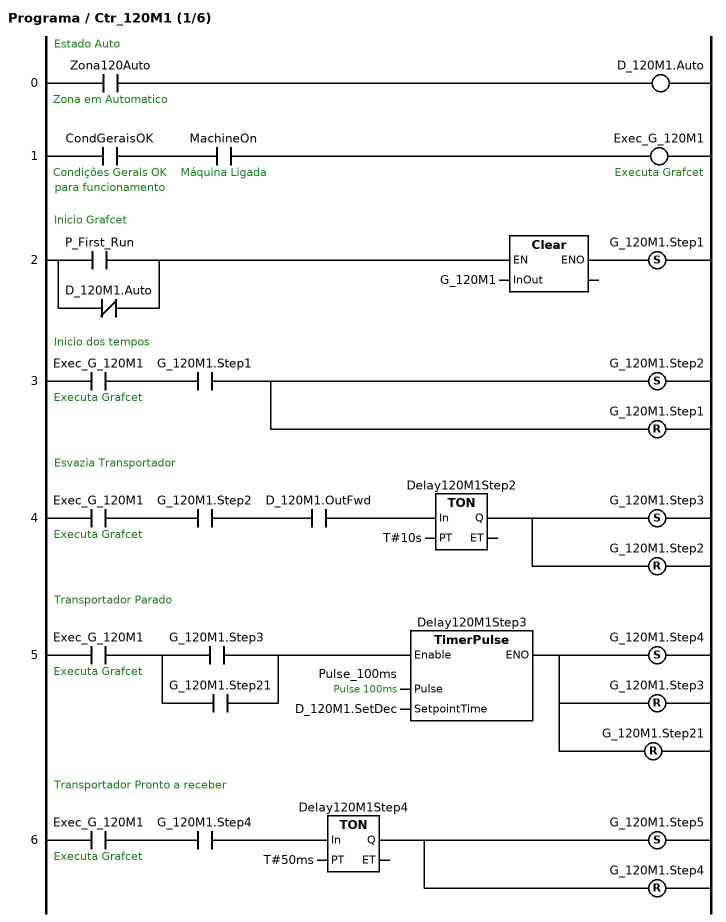
(* [picture p24: Programa / Ctr_120M1, rungs 0-6] *)
(* Rung 0: Estado Auto *)
D_120M1.Auto := Zona120Auto;
(* Rung 1 *)
Exec_G_120M1 := CondGeraisOK AND MachineOn;
(* Rung 2: Inicio Grafcet *)
IF P_First_Run OR NOT D_120M1.Auto THEN
    Clear(InOut := G_120M1);
    G_120M1.Step1 := TRUE;
END_IF;
(* Rung 3: Inicio dos tempos *)
_p41 := Exec_G_120M1 AND G_120M1.Step1;
IF _p41 THEN
    G_120M1.Step2 := TRUE;
    G_120M1.Step1 := FALSE;
END_IF;
(* Rung 4: Esvazia Transportador *)
Delay120M1Step2(In := Exec_G_120M1 AND G_120M1.Step2 AND D_120M1.OutFwd, PT := T#10s);
IF Delay120M1Step2.Q THEN
    G_120M1.Step3 := TRUE;
    G_120M1.Step2 := FALSE;
END_IF;
(* Rung 5: Transportador Parado *)
Delay120M1Step3(Enable := Exec_G_120M1 AND (G_120M1.Step3 OR G_120M1.Step21), Pulse := Pulse_100ms, SetpointTime := D_120M1.SetDec);
IF Delay120M1Step3.ENO THEN
    G_120M1.Step4 := TRUE;
    G_120M1.Step3 := FALSE;
    G_120M1.Step21 := FALSE;
END_IF;
(* Rung 6: Transportador Pronto a receber *)
Delay120M1Step4(In := Exec_G_120M1 AND G_120M1.Step4, PT := T#50ms);
IF Delay120M1Step4.Q THEN
    G_120M1.Step5 := TRUE;
    G_120M1.Step4 := FALSE;
END_IF;

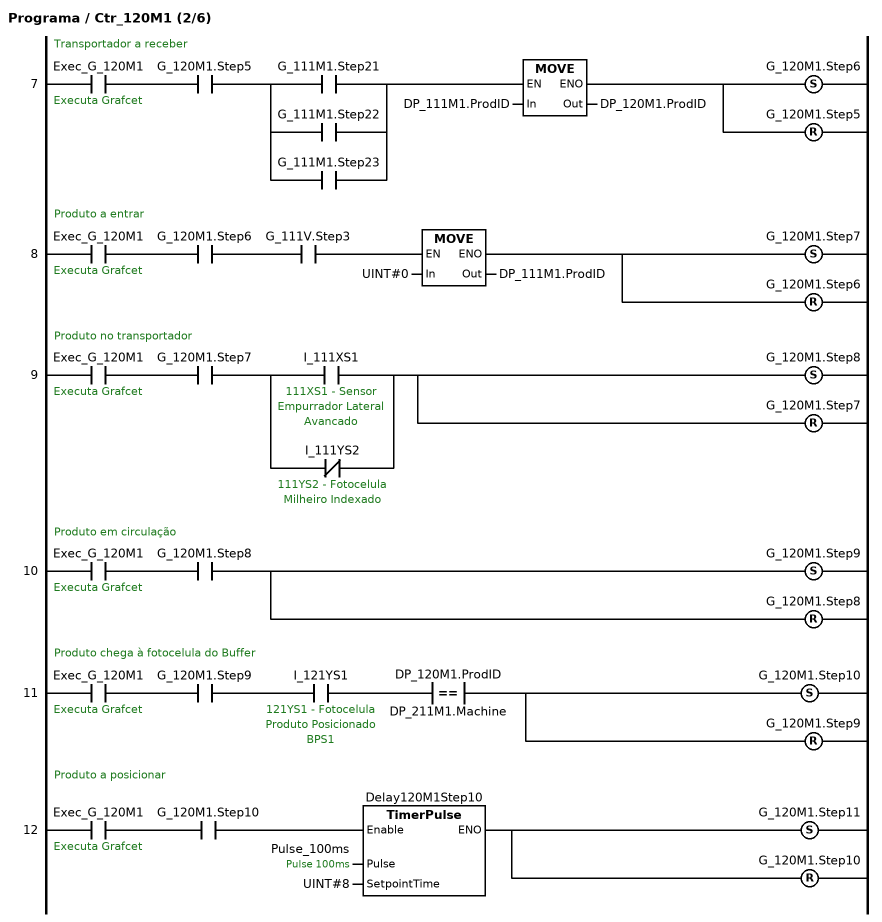
(* Rung 7: Transportador a receber *)
IF Exec_G_120M1 AND G_120M1.Step5 AND (G_111M1.Step21 OR G_111M1.Step22 OR G_111M1.Step23) THEN
    DP_120M1.ProdID := DP_111M1.ProdID;
END_IF;
_p42 := Exec_G_120M1 AND G_120M1.Step5 AND (G_111M1.Step21 OR G_111M1.Step22 OR G_111M1.Step23);
IF _p42 THEN
    G_120M1.Step6 := TRUE;
    G_120M1.Step5 := FALSE;
END_IF;
(* Rung 8: Produto a entrar *)
IF Exec_G_120M1 AND G_120M1.Step6 AND G_111V.Step3 THEN DP_111M1.ProdID := UINT#0; END_IF;
_p43 := Exec_G_120M1 AND G_120M1.Step6 AND G_111V.Step3;
IF _p43 THEN
    G_120M1.Step7 := TRUE;
    G_120M1.Step6 := FALSE;
END_IF;
(* Rung 9: Produto no transportador *)
_p44 := Exec_G_120M1 AND G_120M1.Step7 AND (I_111XS1 OR NOT I_111YS2);
IF _p44 THEN
    G_120M1.Step8 := TRUE;
    G_120M1.Step7 := FALSE;
END_IF;
(* Rung 10: Produto em circulação *)
_p45 := Exec_G_120M1 AND G_120M1.Step8;
IF _p45 THEN
    G_120M1.Step9 := TRUE;
    G_120M1.Step8 := FALSE;
END_IF;
(* Rung 11: Produto chega à fotocelula do Buffer *)
_p46 := Exec_G_120M1 AND G_120M1.Step9 AND I_121YS1 AND (DP_120M1.ProdID = DP_211M1.Machine);
IF _p46 THEN
    G_120M1.Step10 := TRUE;
    G_120M1.Step9 := FALSE;
END_IF;
(* Rung 12: Produto a posicionar *)
Delay120M1Step10(Enable := Exec_G_120M1 AND G_120M1.Step10, Pulse := Pulse_100ms, SetpointTime := UINT#8);
IF Delay120M1Step10.ENO THEN
    G_120M1.Step11 := TRUE;
    G_120M1.Step10 := FALSE;
END_IF;

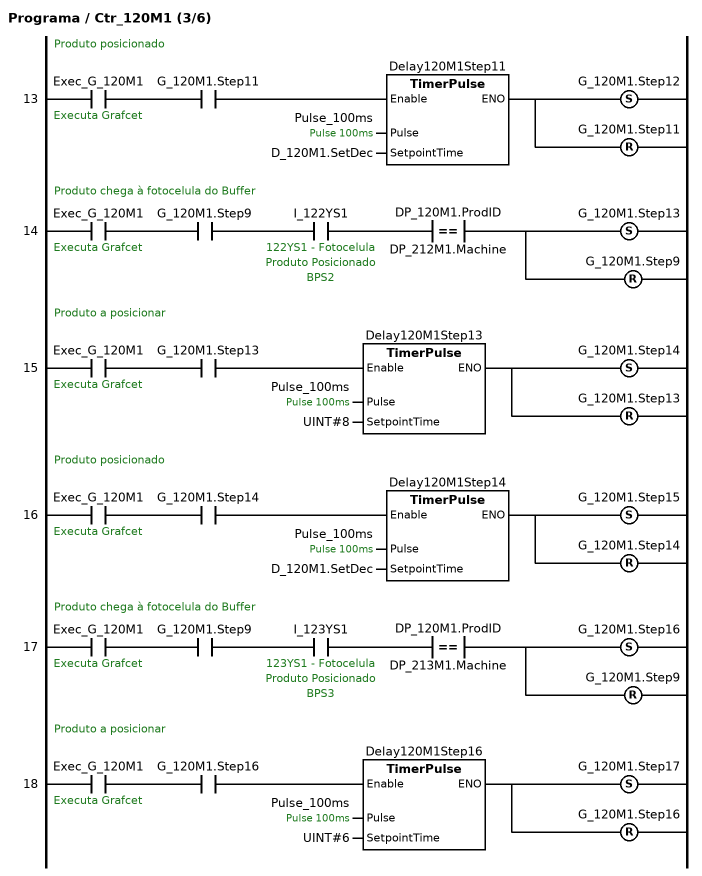
(* Rung 13: Produto posicionado *)
Delay120M1Step11(Enable := Exec_G_120M1 AND G_120M1.Step11, Pulse := Pulse_100ms, SetpointTime := D_120M1.SetDec);
IF Delay120M1Step11.ENO THEN
    G_120M1.Step12 := TRUE;
    G_120M1.Step11 := FALSE;
END_IF;
(* Rung 14: Produto chega à fotocelula do Buffer *)
_p47 := Exec_G_120M1 AND G_120M1.Step9 AND I_122YS1 AND (DP_120M1.ProdID = DP_212M1.Machine);
IF _p47 THEN
    G_120M1.Step13 := TRUE;
    G_120M1.Step9 := FALSE;
END_IF;
(* Rung 15: Produto a posicionar *)
Delay120M1Step13(Enable := Exec_G_120M1 AND G_120M1.Step13, Pulse := Pulse_100ms, SetpointTime := UINT#8);
IF Delay120M1Step13.ENO THEN
    G_120M1.Step14 := TRUE;
    G_120M1.Step13 := FALSE;
END_IF;
(* Rung 16: Produto posicionado *)
Delay120M1Step14(Enable := Exec_G_120M1 AND G_120M1.Step14, Pulse := Pulse_100ms, SetpointTime := D_120M1.SetDec);
IF Delay120M1Step14.ENO THEN
    G_120M1.Step15 := TRUE;
    G_120M1.Step14 := FALSE;
END_IF;
(* Rung 17: Produto chega à fotocelula do Buffer *)
_p48 := Exec_G_120M1 AND G_120M1.Step9 AND I_123YS1 AND (DP_120M1.ProdID = DP_213M1.Machine);
IF _p48 THEN
    G_120M1.Step16 := TRUE;
    G_120M1.Step9 := FALSE;
END_IF;
(* Rung 18: Produto a posicionar *)
Delay120M1Step16(Enable := Exec_G_120M1 AND G_120M1.Step16, Pulse := Pulse_100ms, SetpointTime := UINT#6);
IF Delay120M1Step16.ENO THEN
    G_120M1.Step17 := TRUE;
    G_120M1.Step16 := FALSE;
END_IF;

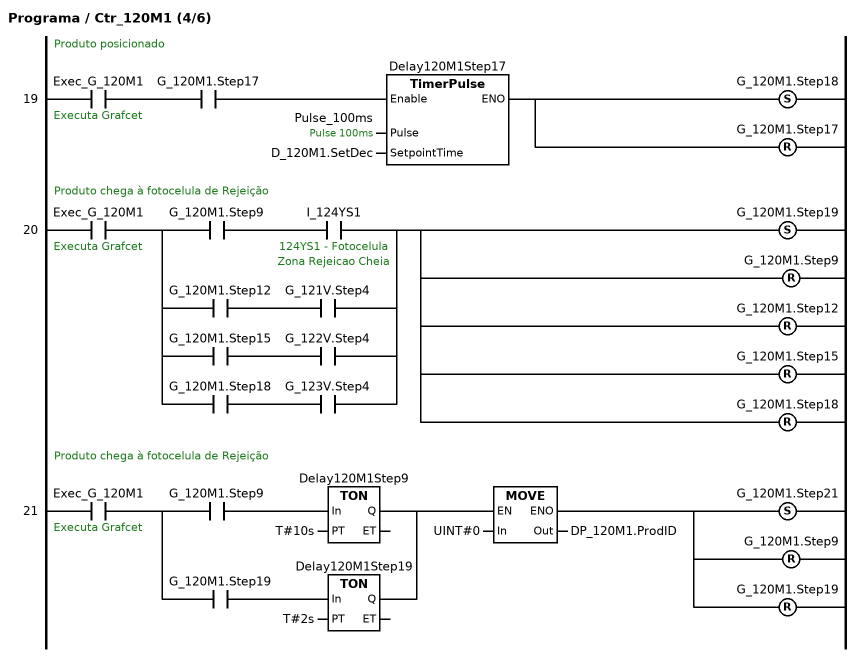
(* Rung 19: Produto posicionado *)
Delay120M1Step17(Enable := Exec_G_120M1 AND G_120M1.Step17, Pulse := Pulse_100ms, SetpointTime := D_120M1.SetDec);
IF Delay120M1Step17.ENO THEN
    G_120M1.Step18 := TRUE;
    G_120M1.Step17 := FALSE;
END_IF;
(* Rung 20: Produto chega à fotocelula de Rejeição *)
_p49 := Exec_G_120M1 AND ((G_120M1.Step9 AND I_124YS1) OR (G_120M1.Step12 AND G_121V.Step4) OR (G_120M1.Step15 AND G_122V.Step4) OR (G_120M1.Step18 AND G_123V.Step4));
IF _p49 THEN
    G_120M1.Step19 := TRUE;
    G_120M1.Step9 := FALSE;
    G_120M1.Step12 := FALSE;
    G_120M1.Step15 := FALSE;
    G_120M1.Step18 := FALSE;
END_IF;
(* Rung 21: Produto chega à fotocelula de Rejeição *)
Delay120M1Step9(In := Exec_G_120M1 AND G_120M1.Step9, PT := T#10s);
Delay120M1Step19(In := Exec_G_120M1 AND G_120M1.Step19, PT := T#2s);
IF Delay120M1Step9.Q OR Delay120M1Step19.Q THEN
    DP_120M1.ProdID := UINT#0;
    G_120M1.Step21 := TRUE;
    G_120M1.Step9 := FALSE;
    G_120M1.Step19 := FALSE;
END_IF;

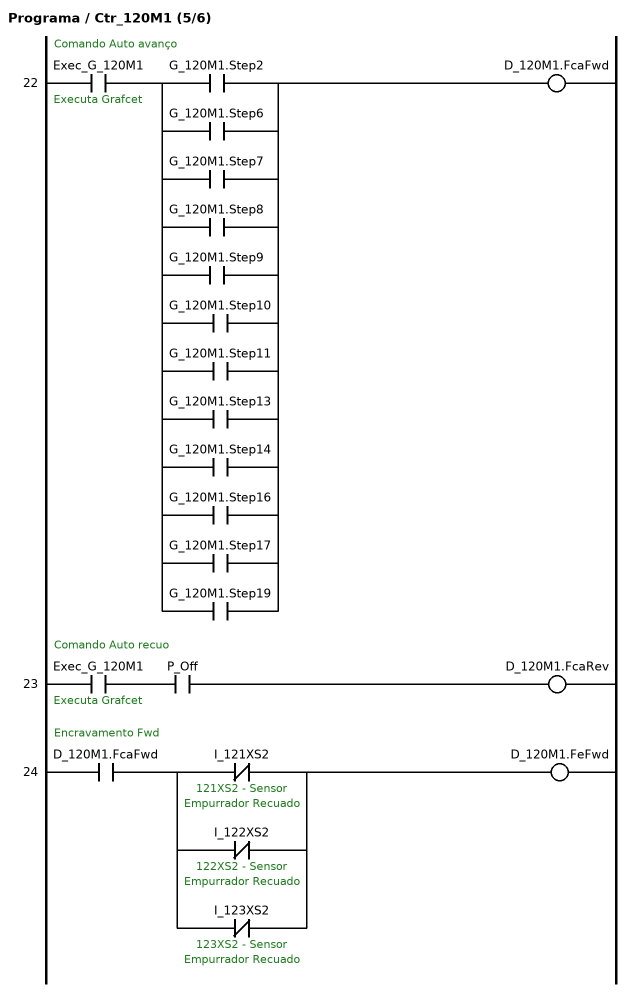
(* Rung 22: Comando Auto avanço *)
D_120M1.FcaFwd := Exec_G_120M1 AND (G_120M1.Step2 OR G_120M1.Step6 OR G_120M1.Step7 OR G_120M1.Step8 OR G_120M1.Step9 OR G_120M1.Step10 OR G_120M1.Step11 OR G_120M1.Step13 OR G_120M1.Step14 OR G_120M1.Step16 OR G_120M1.Step17 OR G_120M1.Step19);
(* Rung 23: Comando Auto recuo *)
D_120M1.FcaRev := Exec_G_120M1 AND P_Off;
(* Rung 24: Encravamento Fwd *)
D_120M1.FeFwd := D_120M1.FcaFwd AND (NOT I_121XS2 OR NOT I_122XS2 OR NOT I_123XS2);

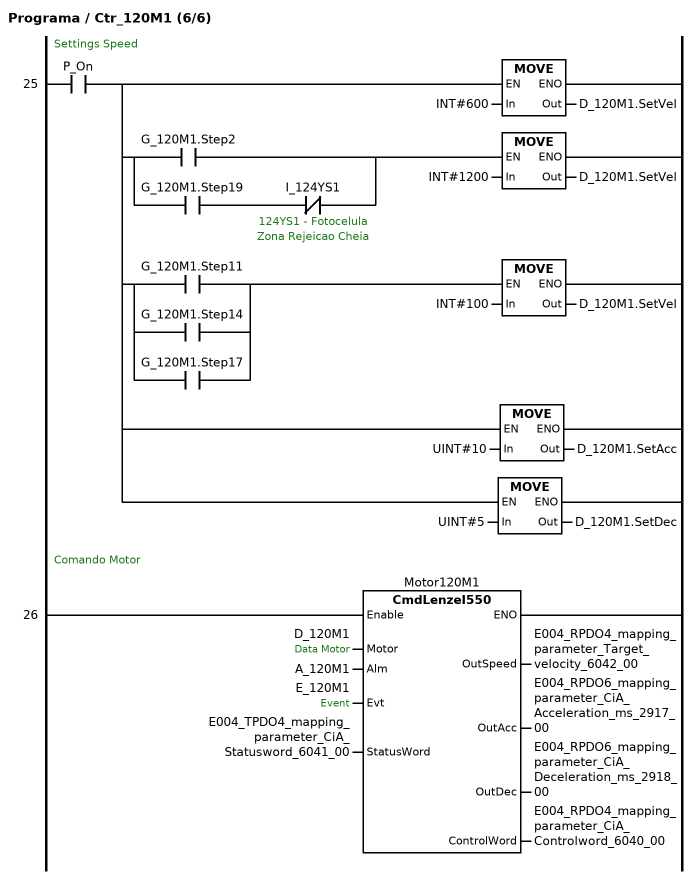
(* Rung 25: Settings Speed *)
IF P_On THEN D_120M1.SetVel := INT#600; END_IF;
IF P_On AND (G_120M1.Step2 OR (G_120M1.Step19 AND NOT I_124YS1)) THEN D_120M1.SetVel := INT#1200; END_IF;
IF P_On AND (G_120M1.Step11 OR G_120M1.Step14 OR G_120M1.Step17) THEN D_120M1.SetVel := INT#100; END_IF;
IF P_On THEN
    D_120M1.SetAcc := UINT#10;
    D_120M1.SetDec := UINT#5;
END_IF;
(* Rung 26: Comando Motor *)
Motor120M1(Enable := TRUE, Motor := D_120M1, Alm := A_120M1, Evt := E_120M1, StatusWord := E004_TPDO4_mapping_parameter_CiA_Statusword_6041_00, OutSpeed => E004_RPDO4_mapping_parameter_Target_velocity_6042_00, OutAcc => E004_RPDO6_mapping_parameter_CiA_Acceleration_ms_2917_00, OutDec => E004_RPDO6_mapping_parameter_CiA_Deceleration_ms_2918_00, ControlWord => E004_RPDO4_mapping_parameter_CiA_Controlword_6040_00);

(* Section Ctr_121V: ladder, written here as Structured Text *)

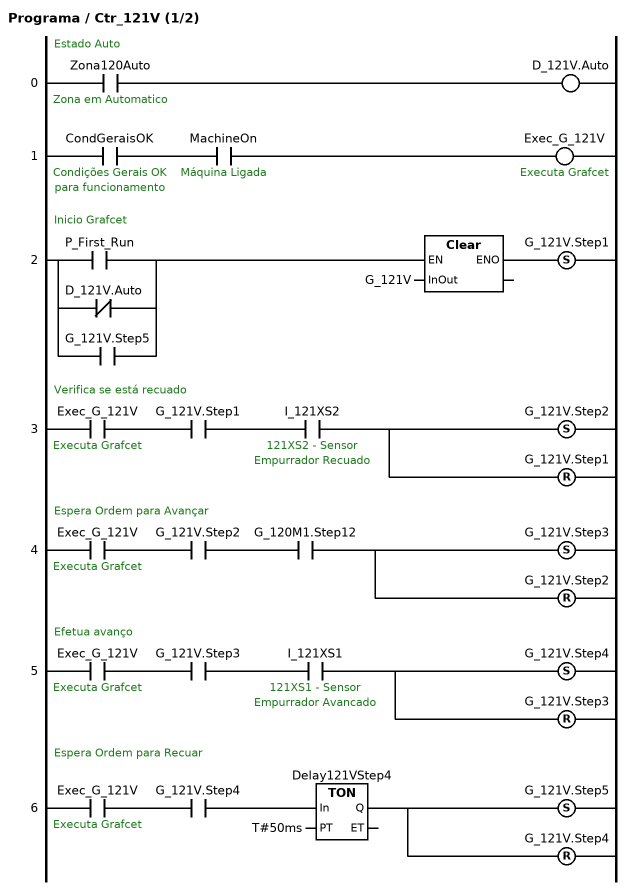
(* Rung 0: Estado Auto *)
D_121V.Auto := Zona120Auto;
(* Rung 1 *)
Exec_G_121V := CondGeraisOK AND MachineOn;
(* Rung 2: Inicio Grafcet *)
_p50 := P_First_Run OR NOT D_121V.Auto OR G_121V.Step5;
IF _p50 THEN
    Clear(InOut := G_121V);
    G_121V.Step1 := TRUE;
END_IF;
(* Rung 3: Verifica se está recuado *)
_p51 := Exec_G_121V AND G_121V.Step1 AND I_121XS2;
IF _p51 THEN
    G_121V.Step2 := TRUE;
    G_121V.Step1 := FALSE;
END_IF;
(* Rung 4: Espera Ordem para Avançar *)
_p52 := Exec_G_121V AND G_121V.Step2 AND G_120M1.Step12;
IF _p52 THEN
    G_121V.Step3 := TRUE;
    G_121V.Step2 := FALSE;
END_IF;
(* Rung 5: Efetua avanço *)
_p53 := Exec_G_121V AND G_121V.Step3 AND I_121XS1;
IF _p53 THEN
    G_121V.Step4 := TRUE;
    G_121V.Step3 := FALSE;
END_IF;
(* Rung 6: Espera Ordem para Recuar *)
Delay121VStep4(In := Exec_G_121V AND G_121V.Step4, PT := T#50ms);
IF Delay121VStep4.Q THEN
    G_121V.Step5 := TRUE;
    G_121V.Step4 := FALSE;
END_IF;

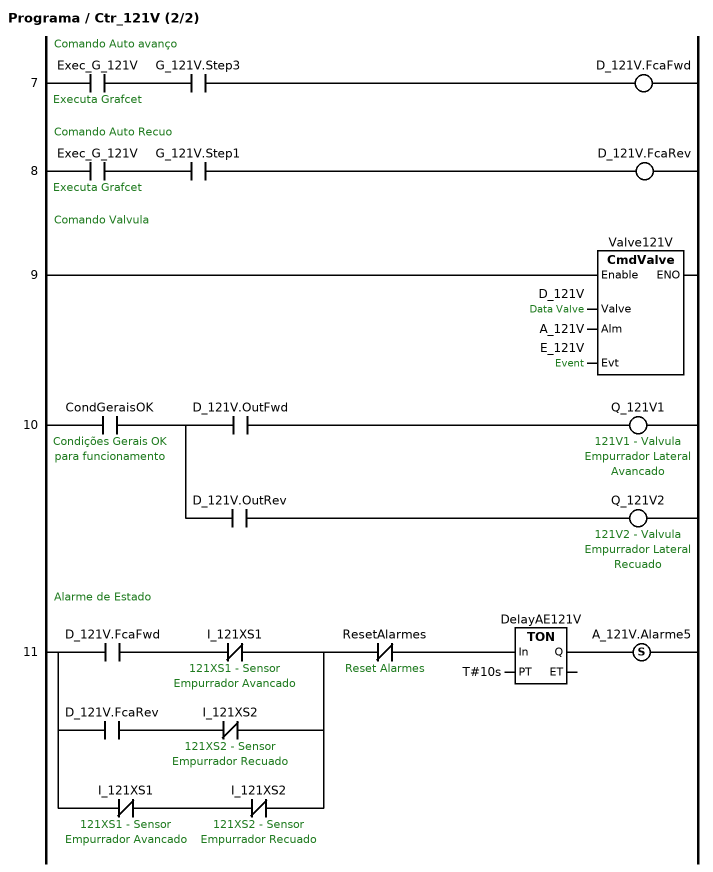
(* Rung 7: Comando Auto avanço *)
D_121V.FcaFwd := Exec_G_121V AND G_121V.Step3;
(* Rung 8: Comando Auto Recuo *)
D_121V.FcaRev := Exec_G_121V AND G_121V.Step1;
(* Rung 9: Comando Valvula *)
Valve121V(Enable := TRUE, Valve := D_121V, Alm := A_121V, Evt := E_121V);
(* Rung 10 *)
Q_121V1 := CondGeraisOK AND D_121V.OutFwd;
Q_121V2 := CondGeraisOK AND D_121V.OutRev;
(* Rung 11: Alarme de Estado *)
DelayAE121V(In := ((D_121V.FcaFwd AND NOT I_121XS1) OR (D_121V.FcaRev AND NOT I_121XS2) OR (NOT I_121XS1 AND NOT I_121XS2)) AND NOT ResetAlarmes, PT := T#10s);
IF DelayAE121V.Q THEN A_121V.Alarme5 := TRUE; END_IF;

(* Section Ctr_122V: ladder, written here as Structured Text *)

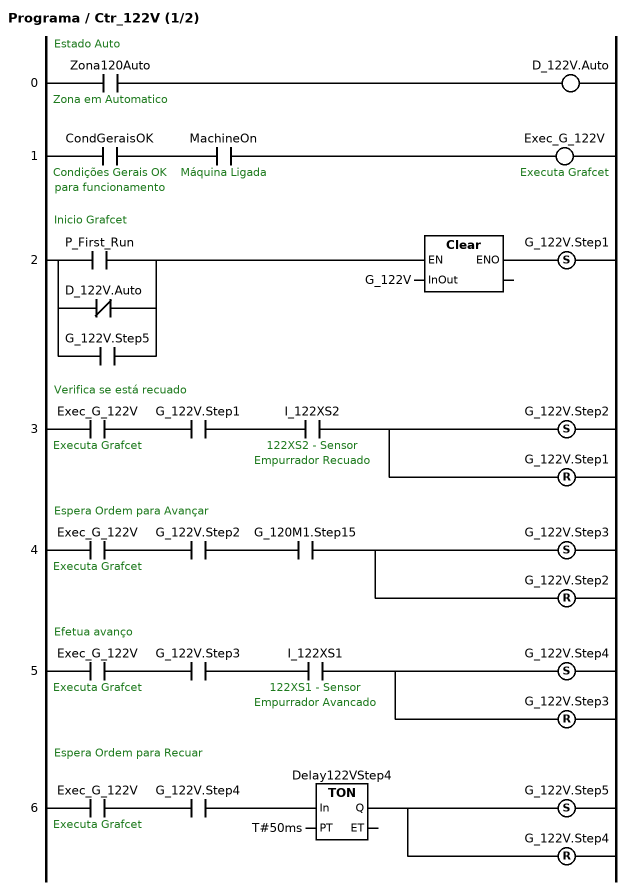
(* Rung 0: Estado Auto *)
D_122V.Auto := Zona120Auto;
(* Rung 1 *)
Exec_G_122V := CondGeraisOK AND MachineOn;
(* Rung 2: Inicio Grafcet *)
_p54 := P_First_Run OR NOT D_122V.Auto OR G_122V.Step5;
IF _p54 THEN
    Clear(InOut := G_122V);
    G_122V.Step1 := TRUE;
END_IF;
(* Rung 3: Verifica se está recuado *)
_p55 := Exec_G_122V AND G_122V.Step1 AND I_122XS2;
IF _p55 THEN
    G_122V.Step2 := TRUE;
    G_122V.Step1 := FALSE;
END_IF;
(* Rung 4: Espera Ordem para Avançar *)
_p56 := Exec_G_122V AND G_122V.Step2 AND G_120M1.Step15;
IF _p56 THEN
    G_122V.Step3 := TRUE;
    G_122V.Step2 := FALSE;
END_IF;
(* Rung 5: Efetua avanço *)
_p57 := Exec_G_122V AND G_122V.Step3 AND I_122XS1;
IF _p57 THEN
    G_122V.Step4 := TRUE;
    G_122V.Step3 := FALSE;
END_IF;
(* Rung 6: Espera Ordem para Recuar *)
Delay122VStep4(In := Exec_G_122V AND G_122V.Step4, PT := T#50ms);
IF Delay122VStep4.Q THEN
    G_122V.Step5 := TRUE;
    G_122V.Step4 := FALSE;
END_IF;

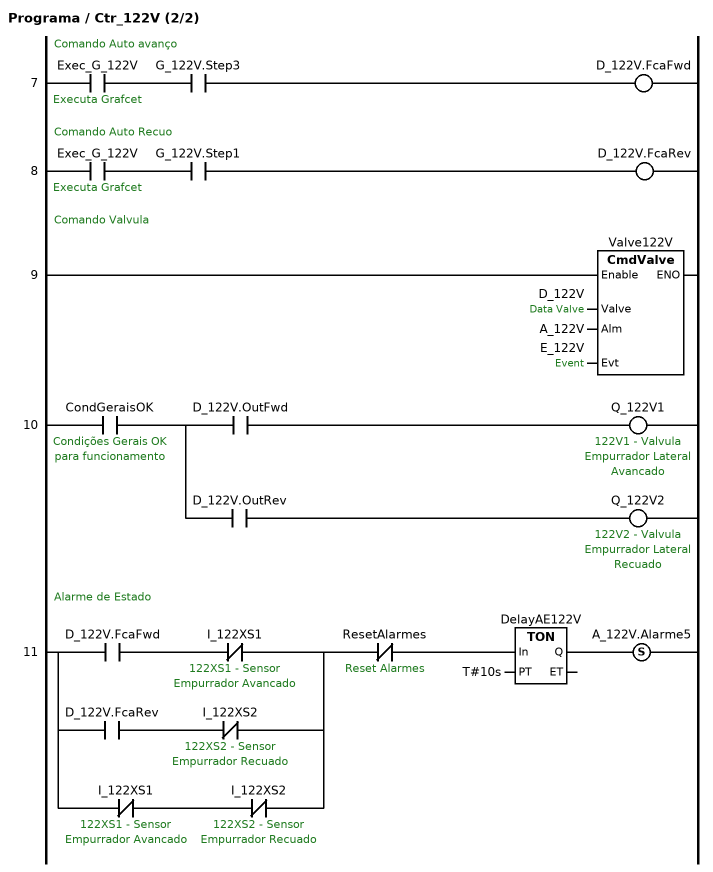
(* Rung 7: Comando Auto avanço *)
D_122V.FcaFwd := Exec_G_122V AND G_122V.Step3;
(* Rung 8: Comando Auto Recuo *)
D_122V.FcaRev := Exec_G_122V AND G_122V.Step1;
(* Rung 9: Comando Valvula *)
Valve122V(Enable := TRUE, Valve := D_122V, Alm := A_122V, Evt := E_122V);
(* Rung 10 *)
Q_122V1 := CondGeraisOK AND D_122V.OutFwd;
Q_122V2 := CondGeraisOK AND D_122V.OutRev;
(* Rung 11: Alarme de Estado *)
DelayAE122V(In := ((D_122V.FcaFwd AND NOT I_122XS1) OR (D_122V.FcaRev AND NOT I_122XS2) OR (NOT I_122XS1 AND NOT I_122XS2)) AND NOT ResetAlarmes, PT := T#10s);
IF DelayAE122V.Q THEN A_122V.Alarme5 := TRUE; END_IF;

(* Section Ctr_123V: ladder, written here as Structured Text *)

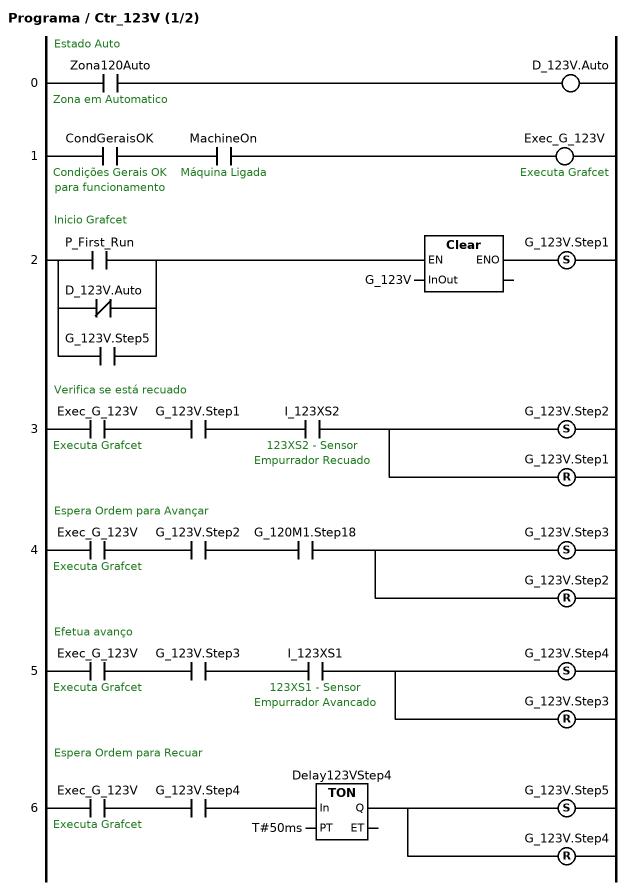
(* Rung 0: Estado Auto *)
D_123V.Auto := Zona120Auto;
(* Rung 1 *)
Exec_G_123V := CondGeraisOK AND MachineOn;
(* Rung 2: Inicio Grafcet *)
_p58 := P_First_Run OR NOT D_123V.Auto OR G_123V.Step5;
IF _p58 THEN
    Clear(InOut := G_123V);
    G_123V.Step1 := TRUE;
END_IF;
(* Rung 3: Verifica se está recuado *)
_p59 := Exec_G_123V AND G_123V.Step1 AND I_123XS2;
IF _p59 THEN
    G_123V.Step2 := TRUE;
    G_123V.Step1 := FALSE;
END_IF;
(* Rung 4: Espera Ordem para Avançar *)
_p60 := Exec_G_123V AND G_123V.Step2 AND G_120M1.Step18;
IF _p60 THEN
    G_123V.Step3 := TRUE;
    G_123V.Step2 := FALSE;
END_IF;
(* Rung 5: Efetua avanço *)
_p61 := Exec_G_123V AND G_123V.Step3 AND I_123XS1;
IF _p61 THEN
    G_123V.Step4 := TRUE;
    G_123V.Step3 := FALSE;
END_IF;
(* Rung 6: Espera Ordem para Recuar *)
Delay123VStep4(In := Exec_G_123V AND G_123V.Step4, PT := T#50ms);
IF Delay123VStep4.Q THEN
    G_123V.Step5 := TRUE;
    G_123V.Step4 := FALSE;
END_IF;

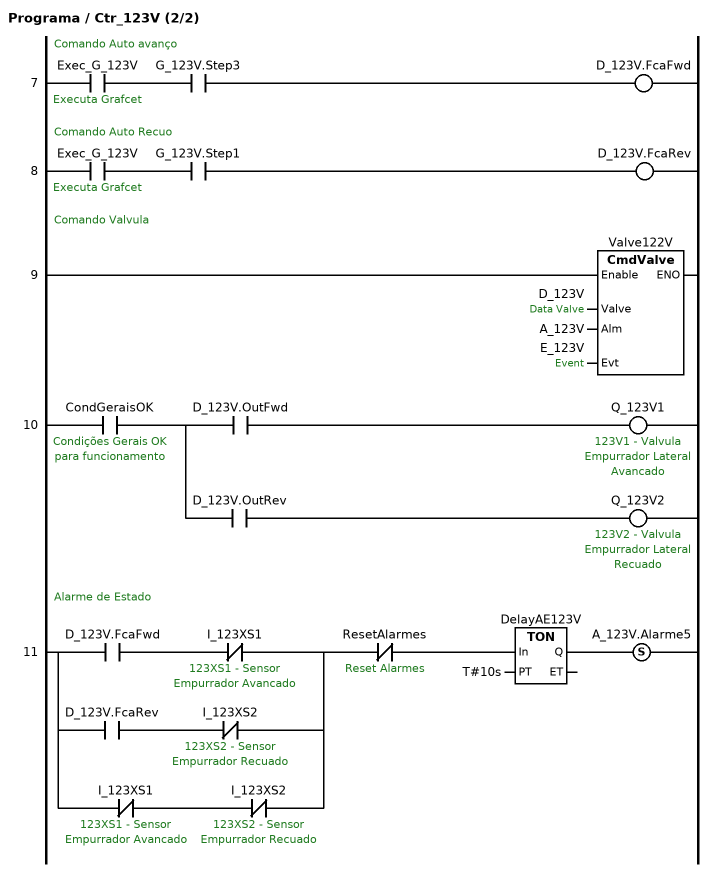
(* Rung 7: Comando Auto avanço *)
D_123V.FcaFwd := Exec_G_123V AND G_123V.Step3;
(* Rung 8: Comando Auto Recuo *)
D_123V.FcaRev := Exec_G_123V AND G_123V.Step1;
(* Rung 9: Comando Valvula *)
Valve122V(Enable := TRUE, Valve := D_123V, Alm := A_123V, Evt := E_123V);
(* Rung 10 *)
Q_123V1 := CondGeraisOK AND D_123V.OutFwd;
Q_123V2 := CondGeraisOK AND D_123V.OutRev;
(* Rung 11: Alarme de Estado *)
DelayAE123V(In := ((D_123V.FcaFwd AND NOT I_123XS1) OR (D_123V.FcaRev AND NOT I_123XS2) OR (NOT I_123XS1 AND NOT I_123XS2)) AND NOT ResetAlarmes, PT := T#10s);
IF DelayAE123V.Q THEN A_123V.Alarme5 := TRUE; END_IF;

(* Section Ctr_211M1: ladder, written here as Structured Text *)

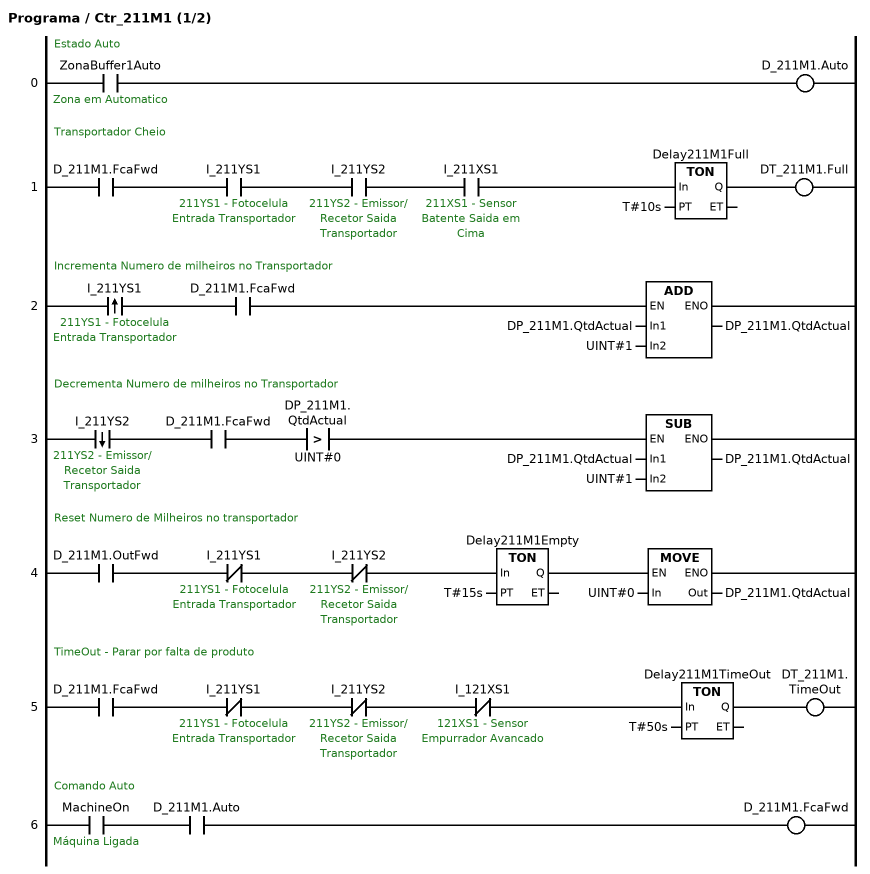
(* Rung 0: Estado Auto *)
D_211M1.Auto := ZonaBuffer1Auto;
(* Rung 1: Transportador Cheio *)
Delay211M1Full(In := D_211M1.FcaFwd AND I_211YS1 AND I_211YS2 AND I_211XS1, PT := T#10s);
DT_211M1.Full := Delay211M1Full.Q;
(* Rung 2: Incrementa Numero de milheiros no Transportador *)
_e62(CLK := I_211YS1);
IF _e62.Q AND D_211M1.FcaFwd THEN DP_211M1.QtdActual := DP_211M1.QtdActual + UINT#1; END_IF;
(* Rung 3: Decrementa Numero de milheiros no Transportador *)
_e63(CLK := I_211YS2);
IF _e63.Q AND D_211M1.FcaFwd AND (DP_211M1.QtdActual > UINT#0) THEN
    DP_211M1.QtdActual := DP_211M1.QtdActual - UINT#1;
END_IF;
(* Rung 4: Reset Numero de Milheiros no transportador *)
Delay211M1Empty(In := D_211M1.OutFwd AND NOT I_211YS1 AND NOT I_211YS2, PT := T#15s);
IF Delay211M1Empty.Q THEN DP_211M1.QtdActual := UINT#0; END_IF;
(* Rung 5: TimeOut - Parar por falta de produto *)
Delay211M1TimeOut(In := D_211M1.FcaFwd AND NOT I_211YS1 AND NOT I_211YS2 AND NOT I_121XS1, PT := T#50s);
DT_211M1.TimeOut := Delay211M1TimeOut.Q;
(* Rung 6: Comando Auto *)
D_211M1.FcaFwd := MachineOn AND D_211M1.Auto;

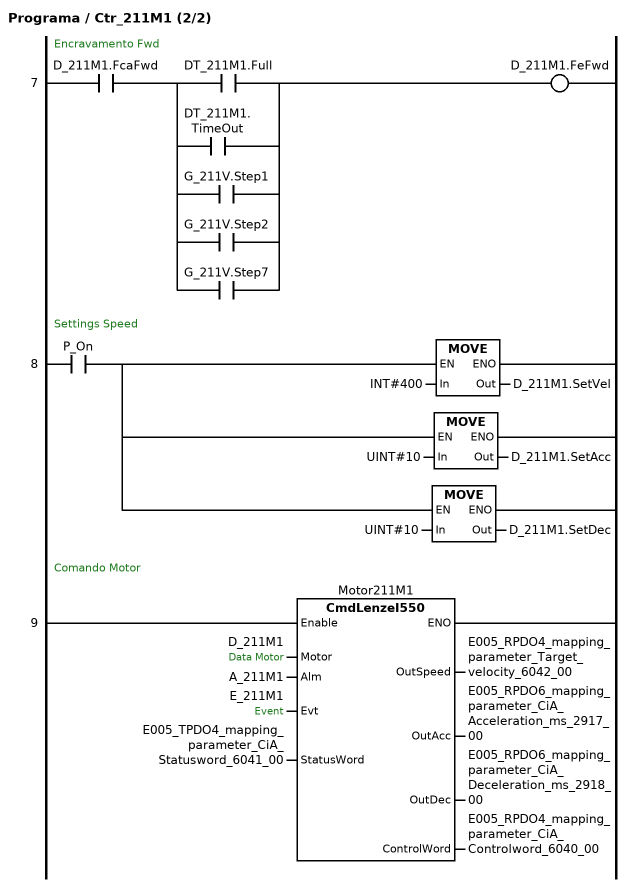
(* Rung 7: Encravamento Fwd *)
D_211M1.FeFwd := D_211M1.FcaFwd AND (DT_211M1.Full OR DT_211M1.TimeOut OR G_211V.Step1 OR G_211V.Step2 OR G_211V.Step7);
(* Rung 8: Settings Speed *)
IF P_On THEN
    D_211M1.SetVel := INT#400;
    D_211M1.SetAcc := UINT#10;
    D_211M1.SetDec := UINT#10;
END_IF;
(* Rung 9: Comando Motor *)
Motor211M1(Enable := TRUE, Motor := D_211M1, Alm := A_211M1, Evt := E_211M1, StatusWord := E005_TPDO4_mapping_parameter_CiA_Statusword_6041_00, OutSpeed => E005_RPDO4_mapping_parameter_Target_velocity_6042_00, OutAcc => E005_RPDO6_mapping_parameter_CiA_Acceleration_ms_2917_00, OutDec => E005_RPDO6_mapping_parameter_CiA_Deceleration_ms_2918_00, ControlWord => E005_RPDO4_mapping_parameter_CiA_Controlword_6040_00);

(* Section Ctr_211V: ladder, written here as Structured Text *)

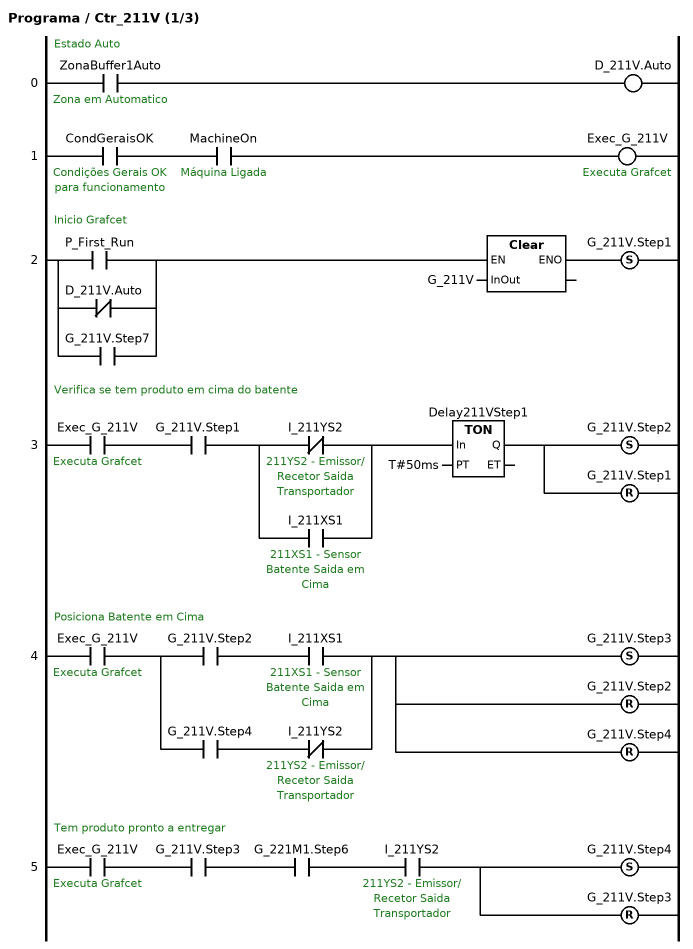
(* Rung 0: Estado Auto *)
D_211V.Auto := ZonaBuffer1Auto;
(* Rung 1 *)
Exec_G_211V := CondGeraisOK AND MachineOn;
(* Rung 2: Inicio Grafcet *)
_p64 := P_First_Run OR NOT D_211V.Auto OR G_211V.Step7;
IF _p64 THEN
    Clear(InOut := G_211V);
    G_211V.Step1 := TRUE;
END_IF;
(* Rung 3: Verifica se tem produto em cima do batente *)
Delay211VStep1(In := Exec_G_211V AND G_211V.Step1 AND (NOT I_211YS2 OR I_211XS1), PT := T#50ms);
IF Delay211VStep1.Q THEN
    G_211V.Step2 := TRUE;
    G_211V.Step1 := FALSE;
END_IF;
(* Rung 4: Posiciona Batente em Cima *)
_p65 := Exec_G_211V AND ((G_211V.Step2 AND I_211XS1) OR (G_211V.Step4 AND NOT I_211YS2));
IF _p65 THEN
    G_211V.Step3 := TRUE;
    G_211V.Step2 := FALSE;
    G_211V.Step4 := FALSE;
END_IF;
(* Rung 5: Tem produto pronto a entregar *)
_p66 := Exec_G_211V AND G_211V.Step3 AND G_221M1.Step6 AND I_211YS2;
IF _p66 THEN
    G_211V.Step4 := TRUE;
    G_211V.Step3 := FALSE;
END_IF;

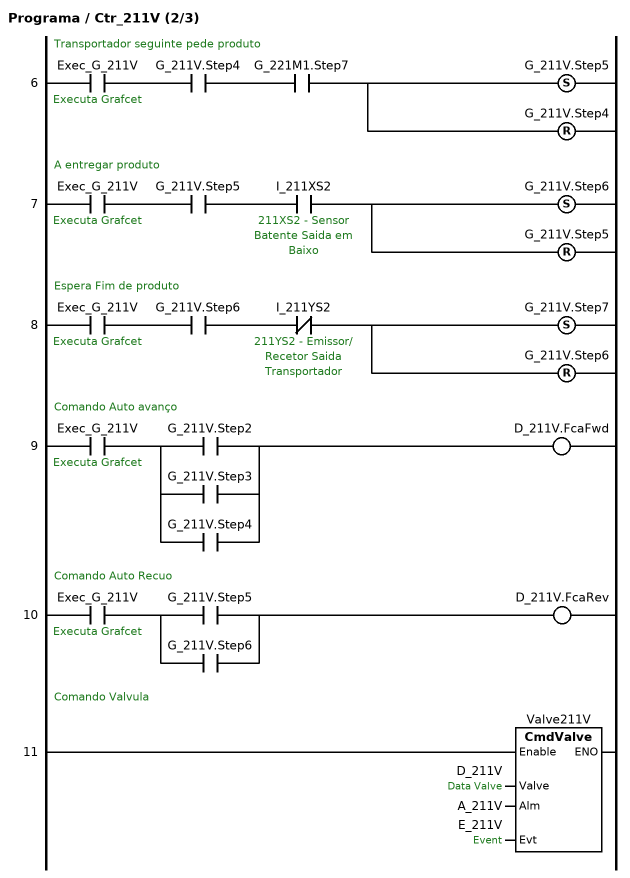
(* Rung 6: Transportador seguinte pede produto *)
_p67 := Exec_G_211V AND G_211V.Step4 AND G_221M1.Step7;
IF _p67 THEN
    G_211V.Step5 := TRUE;
    G_211V.Step4 := FALSE;
END_IF;
(* Rung 7: A entregar produto *)
_p68 := Exec_G_211V AND G_211V.Step5 AND I_211XS2;
IF _p68 THEN
    G_211V.Step6 := TRUE;
    G_211V.Step5 := FALSE;
END_IF;
(* Rung 8: Espera Fim de produto *)
_p69 := Exec_G_211V AND G_211V.Step6 AND NOT I_211YS2;
IF _p69 THEN
    G_211V.Step7 := TRUE;
    G_211V.Step6 := FALSE;
END_IF;
(* Rung 9: Comando Auto avanço *)
D_211V.FcaFwd := Exec_G_211V AND (G_211V.Step2 OR G_211V.Step3 OR G_211V.Step4);
(* Rung 10: Comando Auto Recuo *)
D_211V.FcaRev := Exec_G_211V AND (G_211V.Step5 OR G_211V.Step6);
(* Rung 11: Comando Valvula *)
Valve211V(Enable := TRUE, Valve := D_211V, Alm := A_211V, Evt := E_211V);

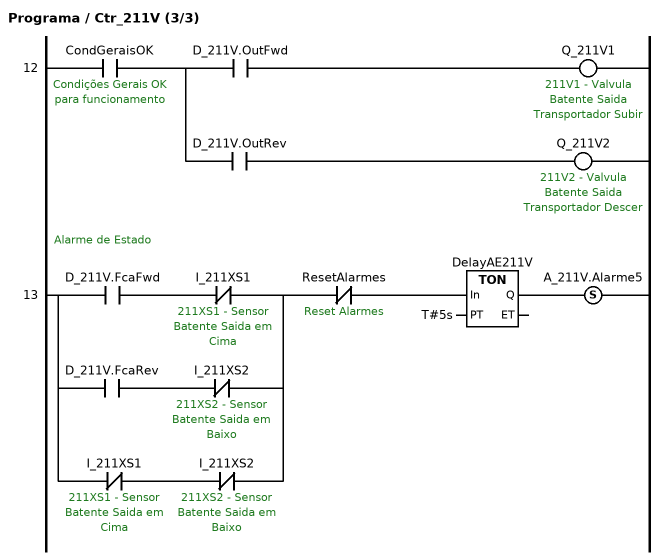
(* Rung 12 *)
Q_211V1 := CondGeraisOK AND D_211V.OutFwd;
Q_211V2 := CondGeraisOK AND D_211V.OutRev;
(* Rung 13: Alarme de Estado *)
DelayAE211V(In := ((D_211V.FcaFwd AND NOT I_211XS1) OR (D_211V.FcaRev AND NOT I_211XS2) OR (NOT I_211XS1 AND NOT I_211XS2)) AND NOT ResetAlarmes, PT := T#5s);
IF DelayAE211V.Q THEN A_211V.Alarme5 := TRUE; END_IF;

(* Section Ctr_212M1: ladder, written here as Structured Text *)

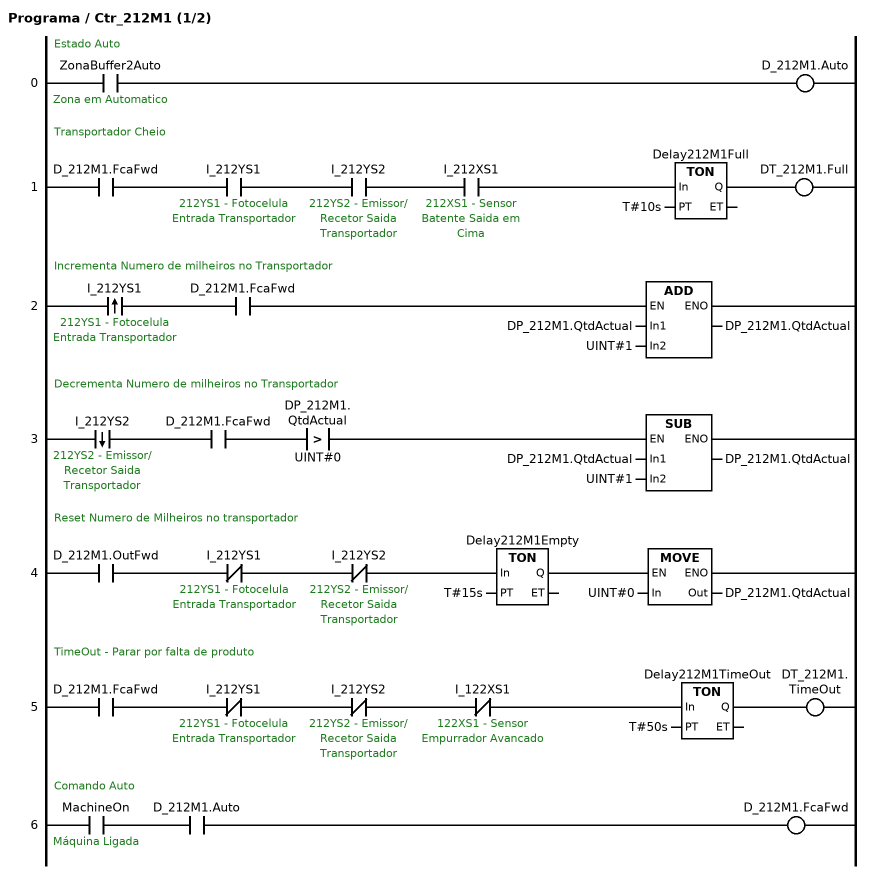
(* Rung 0: Estado Auto *)
D_212M1.Auto := ZonaBuffer2Auto;
(* Rung 1: Transportador Cheio *)
Delay212M1Full(In := D_212M1.FcaFwd AND I_212YS1 AND I_212YS2 AND I_212XS1, PT := T#10s);
DT_212M1.Full := Delay212M1Full.Q;
(* Rung 2: Incrementa Numero de milheiros no Transportador *)
_e70(CLK := I_212YS1);
IF _e70.Q AND D_212M1.FcaFwd THEN DP_212M1.QtdActual := DP_212M1.QtdActual + UINT#1; END_IF;
(* Rung 3: Decrementa Numero de milheiros no Transportador *)
_e71(CLK := I_212YS2);
IF _e71.Q AND D_212M1.FcaFwd AND (DP_212M1.QtdActual > UINT#0) THEN
    DP_212M1.QtdActual := DP_212M1.QtdActual - UINT#1;
END_IF;
(* Rung 4: Reset Numero de Milheiros no transportador *)
Delay212M1Empty(In := D_212M1.OutFwd AND NOT I_212YS1 AND NOT I_212YS2, PT := T#15s);
IF Delay212M1Empty.Q THEN DP_212M1.QtdActual := UINT#0; END_IF;
(* Rung 5: TimeOut - Parar por falta de produto *)
Delay212M1TimeOut(In := D_212M1.FcaFwd AND NOT I_212YS1 AND NOT I_212YS2 AND NOT I_122XS1, PT := T#50s);
DT_212M1.TimeOut := Delay212M1TimeOut.Q;
(* Rung 6: Comando Auto *)
D_212M1.FcaFwd := MachineOn AND D_212M1.Auto;

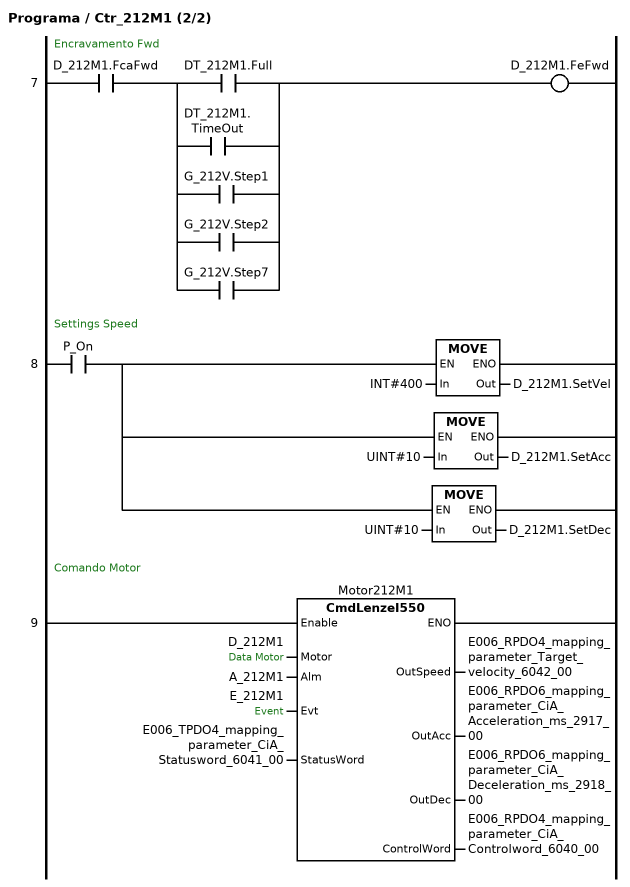
(* Rung 7: Encravamento Fwd *)
D_212M1.FeFwd := D_212M1.FcaFwd AND (DT_212M1.Full OR DT_212M1.TimeOut OR G_212V.Step1 OR G_212V.Step2 OR G_212V.Step7);
(* Rung 8: Settings Speed *)
IF P_On THEN
    D_212M1.SetVel := INT#400;
    D_212M1.SetAcc := UINT#10;
    D_212M1.SetDec := UINT#10;
END_IF;
(* Rung 9: Comando Motor *)
Motor212M1(Enable := TRUE, Motor := D_212M1, Alm := A_212M1, Evt := E_212M1, StatusWord := E006_TPDO4_mapping_parameter_CiA_Statusword_6041_00, OutSpeed => E006_RPDO4_mapping_parameter_Target_velocity_6042_00, OutAcc => E006_RPDO6_mapping_parameter_CiA_Acceleration_ms_2917_00, OutDec => E006_RPDO6_mapping_parameter_CiA_Deceleration_ms_2918_00, ControlWord => E006_RPDO4_mapping_parameter_CiA_Controlword_6040_00);

(* Section Ctr_212V: ladder, written here as Structured Text *)

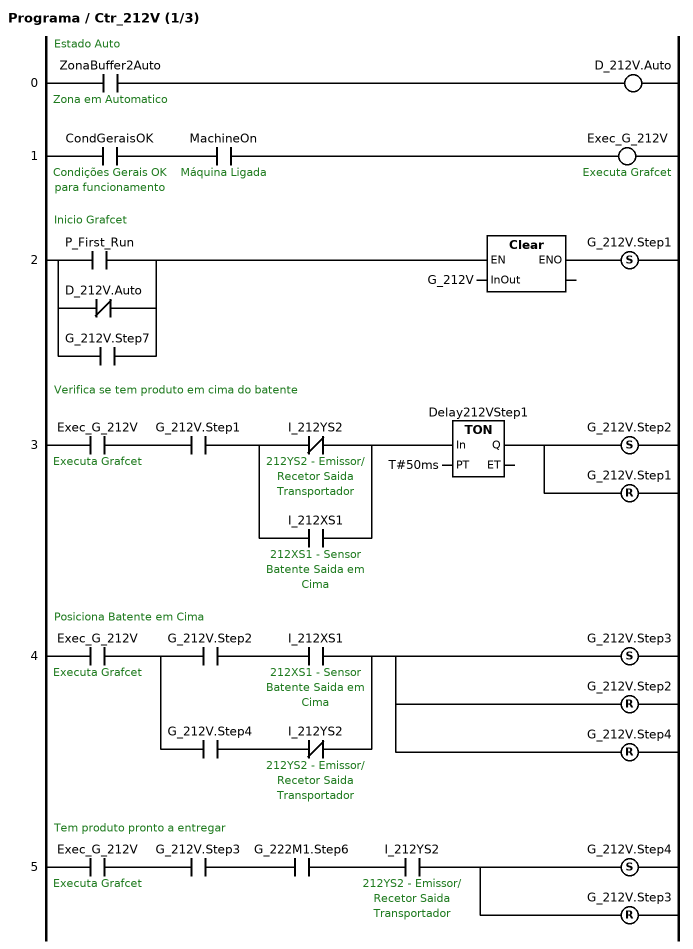
(* Rung 0: Estado Auto *)
D_212V.Auto := ZonaBuffer2Auto;
(* Rung 1 *)
Exec_G_212V := CondGeraisOK AND MachineOn;
(* Rung 2: Inicio Grafcet *)
_p72 := P_First_Run OR NOT D_212V.Auto OR G_212V.Step7;
IF _p72 THEN
    Clear(InOut := G_212V);
    G_212V.Step1 := TRUE;
END_IF;
(* Rung 3: Verifica se tem produto em cima do batente *)
Delay212VStep1(In := Exec_G_212V AND G_212V.Step1 AND (NOT I_212YS2 OR I_212XS1), PT := T#50ms);
IF Delay212VStep1.Q THEN
    G_212V.Step2 := TRUE;
    G_212V.Step1 := FALSE;
END_IF;
(* Rung 4: Posiciona Batente em Cima *)
_p73 := Exec_G_212V AND ((G_212V.Step2 AND I_212XS1) OR (G_212V.Step4 AND NOT I_212YS2));
IF _p73 THEN
    G_212V.Step3 := TRUE;
    G_212V.Step2 := FALSE;
    G_212V.Step4 := FALSE;
END_IF;
(* Rung 5: Tem produto pronto a entregar *)
_p74 := Exec_G_212V AND G_212V.Step3 AND G_222M1.Step6 AND I_212YS2;
IF _p74 THEN
    G_212V.Step4 := TRUE;
    G_212V.Step3 := FALSE;
END_IF;

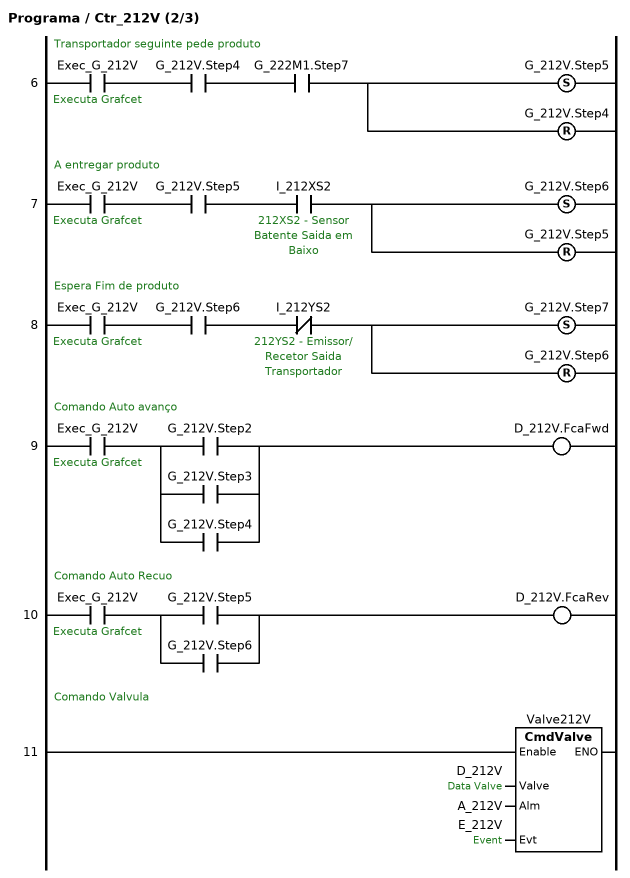
(* Rung 6: Transportador seguinte pede produto *)
_p75 := Exec_G_212V AND G_212V.Step4 AND G_222M1.Step7;
IF _p75 THEN
    G_212V.Step5 := TRUE;
    G_212V.Step4 := FALSE;
END_IF;
(* Rung 7: A entregar produto *)
_p76 := Exec_G_212V AND G_212V.Step5 AND I_212XS2;
IF _p76 THEN
    G_212V.Step6 := TRUE;
    G_212V.Step5 := FALSE;
END_IF;
(* Rung 8: Espera Fim de produto *)
_p77 := Exec_G_212V AND G_212V.Step6 AND NOT I_212YS2;
IF _p77 THEN
    G_212V.Step7 := TRUE;
    G_212V.Step6 := FALSE;
END_IF;
(* Rung 9: Comando Auto avanço *)
D_212V.FcaFwd := Exec_G_212V AND (G_212V.Step2 OR G_212V.Step3 OR G_212V.Step4);
(* Rung 10: Comando Auto Recuo *)
D_212V.FcaRev := Exec_G_212V AND (G_212V.Step5 OR G_212V.Step6);
(* Rung 11: Comando Valvula *)
Valve212V(Enable := TRUE, Valve := D_212V, Alm := A_212V, Evt := E_212V);

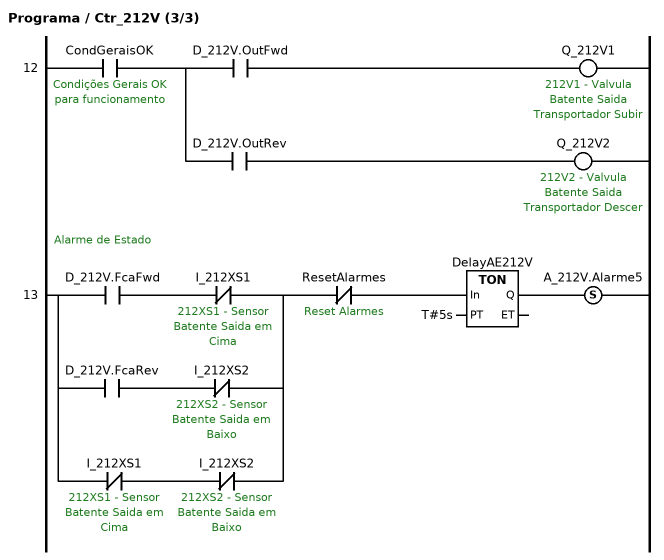
(* Rung 12 *)
Q_212V1 := CondGeraisOK AND D_212V.OutFwd;
Q_212V2 := CondGeraisOK AND D_212V.OutRev;
(* Rung 13: Alarme de Estado *)
DelayAE212V(In := ((D_212V.FcaFwd AND NOT I_212XS1) OR (D_212V.FcaRev AND NOT I_212XS2) OR (NOT I_212XS1 AND NOT I_212XS2)) AND NOT ResetAlarmes, PT := T#5s);
IF DelayAE212V.Q THEN A_212V.Alarme5 := TRUE; END_IF;

(* Section Ctr_213M1: ladder, written here as Structured Text *)

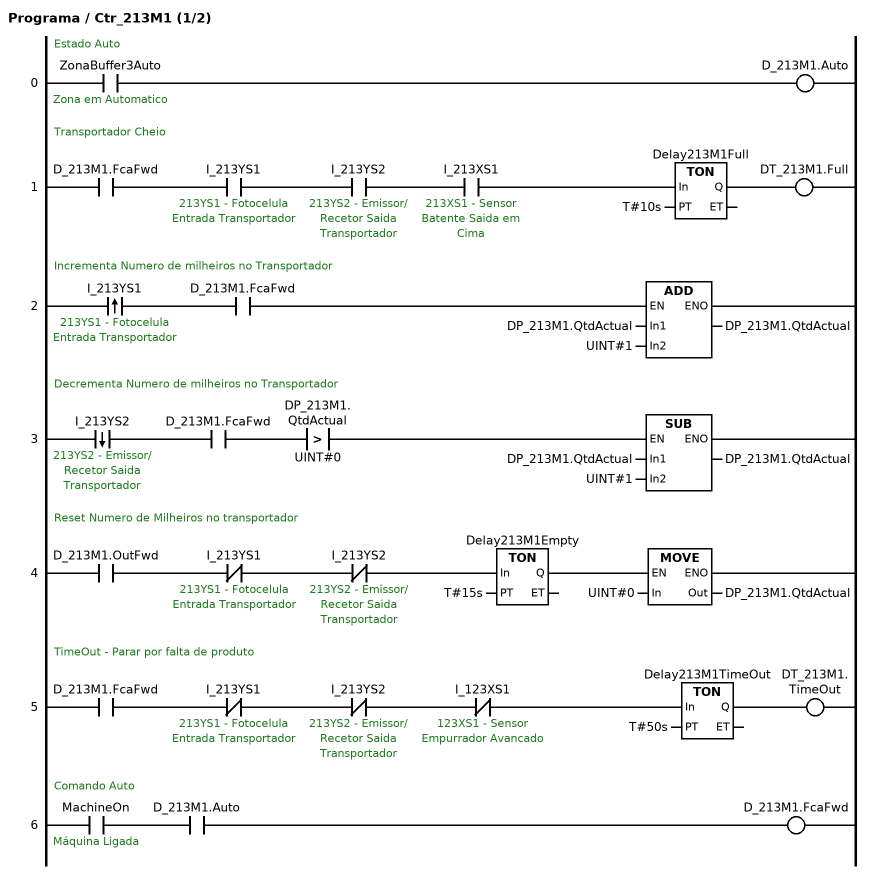
(* Rung 0: Estado Auto *)
D_213M1.Auto := ZonaBuffer3Auto;
(* Rung 1: Transportador Cheio *)
Delay213M1Full(In := D_213M1.FcaFwd AND I_213YS1 AND I_213YS2 AND I_213XS1, PT := T#10s);
DT_213M1.Full := Delay213M1Full.Q;
(* Rung 2: Incrementa Numero de milheiros no Transportador *)
_e78(CLK := I_213YS1);
IF _e78.Q AND D_213M1.FcaFwd THEN DP_213M1.QtdActual := DP_213M1.QtdActual + UINT#1; END_IF;
(* Rung 3: Decrementa Numero de milheiros no Transportador *)
_e79(CLK := I_213YS2);
IF _e79.Q AND D_213M1.FcaFwd AND (DP_213M1.QtdActual > UINT#0) THEN
    DP_213M1.QtdActual := DP_213M1.QtdActual - UINT#1;
END_IF;
(* Rung 4: Reset Numero de Milheiros no transportador *)
Delay213M1Empty(In := D_213M1.OutFwd AND NOT I_213YS1 AND NOT I_213YS2, PT := T#15s);
IF Delay213M1Empty.Q THEN DP_213M1.QtdActual := UINT#0; END_IF;
(* Rung 5: TimeOut - Parar por falta de produto *)
Delay213M1TimeOut(In := D_213M1.FcaFwd AND NOT I_213YS1 AND NOT I_213YS2 AND NOT I_123XS1, PT := T#50s);
DT_213M1.TimeOut := Delay213M1TimeOut.Q;
(* Rung 6: Comando Auto *)
D_213M1.FcaFwd := MachineOn AND D_213M1.Auto;

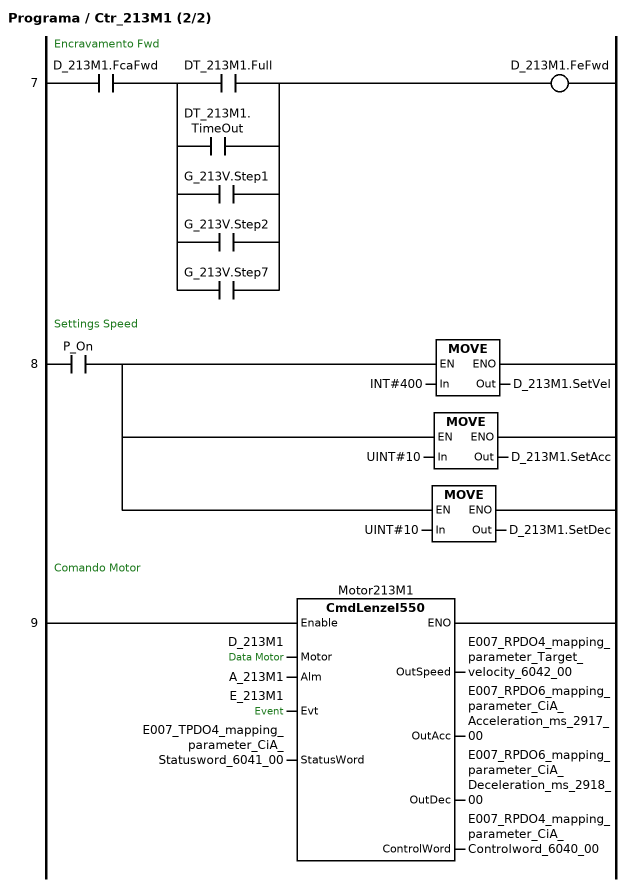
(* Rung 7: Encravamento Fwd *)
D_213M1.FeFwd := D_213M1.FcaFwd AND (DT_213M1.Full OR DT_213M1.TimeOut OR G_213V.Step1 OR G_213V.Step2 OR G_213V.Step7);
(* Rung 8: Settings Speed *)
IF P_On THEN
    D_213M1.SetVel := INT#400;
    D_213M1.SetAcc := UINT#10;
    D_213M1.SetDec := UINT#10;
END_IF;
(* Rung 9: Comando Motor *)
Motor213M1(Enable := TRUE, Motor := D_213M1, Alm := A_213M1, Evt := E_213M1, StatusWord := E007_TPDO4_mapping_parameter_CiA_Statusword_6041_00, OutSpeed => E007_RPDO4_mapping_parameter_Target_velocity_6042_00, OutAcc => E007_RPDO6_mapping_parameter_CiA_Acceleration_ms_2917_00, OutDec => E007_RPDO6_mapping_parameter_CiA_Deceleration_ms_2918_00, ControlWord => E007_RPDO4_mapping_parameter_CiA_Controlword_6040_00);

(* Section Ctr_213V: ladder, written here as Structured Text *)

